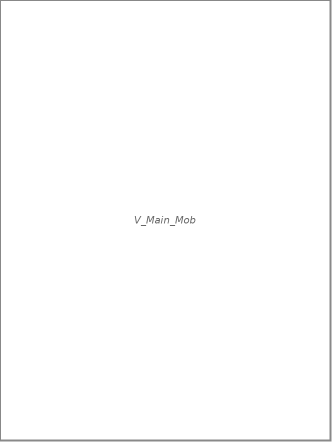
VISUALIZATION VisuStart  // 332x442
    Frame (0,0 330x440)
        shows V_Main_Mob()
END_VISUALIZATION

(* stored: Version 1.1.0.1, ProductVersion 3.1.4018.5
   Visu VisuStart: Id {d6686b52-89fb-44b4-9d64-392408488888} *)
